LIN {X 0,Y 130.149,Z 483.599,A -85,B 0,C 180,E1 -28284.751,E2 -28284.751} C_VEL
LIN {X 0,Y 128.959,Z 485.397,A -85,B 0,C 180,E1 -28285.729,E2 -28285.729} C_VEL
LIN {X 0,Y 120.311,Z 494.144,A -85,B 0,C 180,E1 -28288.807,E2 -28288.807} C_VEL
LIN {X 0,Y 110.679,Z 502.592,A -85,B 0,C 180,E1 -28292.714,E2 -28292.714} C_VEL
LIN {X 0,Y 101.639,Z 509.611,A -85,B 0,C 180,E1 -28297.325,E2 -28297.325} C_VEL
LIN {X 0,Y 92.583,Z 515.883,A -85,B 0,C 180,E1 -28303.336,E2 -28303.336} C_VEL
LIN {X 0,Y 84.526,Z 520.929,A -85,B 0,C 180,E1 -28310.77,E2 -28310.77} C_VEL
LIN {X 0,Y 81.105,Z 522.68,A -85,B 0,C 180,E1 -28313.879,E2 -28313.879} C_VEL
LIN {X 0,Y 74.401,Z 525.173,A -85,B 0,C 180,E1 -28318.954,E2 -28318.954} C_VEL
LIN {X 0,Y 69.318,Z 526.805,A -85,B 0,C 180,E1 -28323.682,E2 -28323.682} C_VEL
LIN {X 0,Y 66.499,Z 527.76,A -85,B 0,C 180,E1 -28328.01,E2 -28328.01} C_VEL
LIN {X 0,Y 65.882,Z 527.988,A -85,B 0,C 180,E1 -28329.615,E2 -28329.615} C_VEL
LIN {X 0,Y 64.073,Z 528.951,A -85,B 0,C 180,E1 -28337.325,E2 -28337.325} C_VEL
LIN {X 0,Y 63.109,Z 529.528,A -85,B 0,C 180,E1 -28349.997,E2 -28349.997} C_VEL
LIN {X 0,Y 64.071,Z 528.979,A -85,B 0,C 180,E1 -28362.67,E2 -28362.67} C_VEL
LIN {X 0,Y 67.407,Z 527.331,A -85,B 0,C 180,E1 -28374.645,E2 -28374.645} C_VEL
LIN {X 0,Y 73.03,Z 524.535,A -85,B 0,C 180,E1 -28385.265,E2 -28385.265} C_VEL
LIN {X 0,Y 80.719,Z 520.508,A -85,B 0,C 180,E1 -28394.147,E2 -28394.147} C_VEL
LIN {X 0,Y 89.779,Z 515.164,A -85,B 0,C 180,E1 -28401.515,E2 -28401.515} C_VEL
LIN {X 0,Y 100.079,Z 508.331,A -85,B 0,C 180,E1 -28407.423,E2 -28407.423} C_VEL
LIN {X 0,Y 111.151,Z 499.793,A -85,B 0,C 180,E1 -28412.273,E2 -28412.273} C_VEL
LIN {X 0,Y 119.919,Z 492.105,A -85,B 0,C 180,E1 -28415.281,E2 -28415.281} C_VEL
LIN {X 0,Y 124.065,Z 488.02,A -85,B 0,C 180,E1 -28416.638,E2 -28416.638} C_VEL
LIN {X 0,Y 125.032,Z 486.59,A -85,B 0,C 180,E1 -28417.702,E2 -28417.702} C_VEL
LIN {X 0,Y 125.654,Z 484.374,A -85,B 0,C 180,E1 -28420.391,E2 -28420.391} C_VEL
LIN {X 0,Y 126.101,Z 482.181,A -85,B 0,C 180,E1 -28423.819,E2 -28423.819} C_VEL
LIN {X 0,Y 126.419,Z 480.387,A -85,B 0,C 180,E1 -28427.151,E2 -28427.151} C_VEL
LIN {X 0,Y 126.751,Z 478.972,A -85,B 0,C 180,E1 -28430.424,E2 -28430.424} C_VEL
LIN {X 0,Y 127.15,Z 477.836,A -85,B 0,C 180,E1 -28434.208,E2 -28434.208} C_VEL
LIN {X 0,Y 127.894,Z 476.973,A -85,B 0,C 180,E1 -28440,E2 -28440} C_VEL
LIN {X 0,Y 127.63,Z 477.823,A -85,B 0,C 180,E1 -28443.156,E2 -28443.156} C_VEL
LIN {X 0,Y 127.297,Z 479.151,A -85,B 0,C 180,E1 -28446.411,E2 -28446.411} C_VEL
LIN {X 0,Y 126.775,Z 480.998,A -85,B 0,C 180,E1 -28449.573,E2 -28449.573} C_VEL
LIN {X 0,Y 125.931,Z 483.628,A -85,B 0,C 180,E1 -28452.899,E2 -28452.899} C_VEL
LIN {X 0,Y 124.857,Z 486.8,A -85,B 0,C 180,E1 -28456.346,E2 -28456.346} C_VEL
LIN {X 0,Y 123.396,Z 490.697,A -85,B 0,C 180,E1 -28459.982,E2 -28459.982} C_VEL
LIN {X 0,Y 121.154,Z 493.836,A -85,B 0,C 180,E1 -28461.858,E2 -28461.858} C_VEL
LIN {X 0,Y 112.191,Z 502.139,A -85,B 0,C 180,E1 -28464.729,E2 -28464.729} C_VEL
LIN {X 0,Y 103.535,Z 509.243,A -85,B 0,C 180,E1 -28468.065,E2 -28468.065} C_VEL
LIN {X 0,Y 92.735,Z 517.125,A -85,B 0,C 180,E1 -28473.528,E2 -28473.528} C_VEL
LIN {X 0,Y 82.856,Z 523.405,A -85,B 0,C 180,E1 -28480.239,E2 -28480.239} C_VEL
LIN {X 0,Y 73.58,Z 528.827,A -85,B 0,C 180,E1 -28489.828,E2 -28489.828} C_VEL
LIN {X 0,Y 68.028,Z 531.891,A -85,B 0,C 180,E1 -28498.902,E2 -28498.902} C_VEL
LIN {X 0,Y 63.951,Z 534.284,A -85,B 0,C 180,E1 -28510.753,E2 -28510.753} C_VEL
LIN {X 0,Y 62.616,Z 535.521,A -85,B 0,C 180,E1 -28523.558,E2 -28523.558} C_VEL
LIN {X 0,Y 62.844,Z 535.701,A -85,B 0,C 180,E1 -28530.003,E2 -28530.003} C_VEL
LIN {X 0,Y 62.959,Z 535.026,A -85,B 0,C 180,E1 -28542.903,E2 -28542.903} C_VEL
LIN {X 0,Y 65.625,Z 533.183,A -85,B 0,C 180,E1 -28555.367,E2 -28555.367} C_VEL
LIN {X 0,Y 70.963,Z 530.169,A -85,B 0,C 180,E1 -28566.46,E2 -28566.46} C_VEL
LIN {X 0,Y 78.454,Z 525.917,A -85,B 0,C 180,E1 -28575.782,E2 -28575.782} C_VEL
LIN {X 0,Y 87.629,Z 520.319,A -85,B 0,C 180,E1 -28583.327,E2 -28583.327} C_VEL
LIN {X 0,Y 98.045,Z 513.228,A -85,B 0,C 180,E1 -28589.34,E2 -28589.34} C_VEL
LIN {X 0,Y 107.812,Z 505.657,A -85,B 0,C 180,E1 -28593.683,E2 -28593.683} C_VEL
LIN {X 0,Y 118.2,Z 496.56,A -85,B 0,C 180,E1 -28597.166,E2 -28597.166} C_VEL
LIN {X 0,Y 121.117,Z 493.584,A -85,B 0,C 180,E1 -28598.194,E2 -28598.194} C_VEL
LIN {X 0,Y 123.249,Z 490.578,A -85,B 0,C 180,E1 -28599.993,E2 -28599.993} C_VEL
LIN {X 0,Y 124.755,Z 486.626,A -85,B 0,C 180,E1 -28603.64,E2 -28603.64} C_VEL
LIN {X 0,Y 125.861,Z 483.397,A -85,B 0,C 180,E1 -28607.094,E2 -28607.094} C_VEL
LIN {X 0,Y 126.654,Z 480.815,A -85,B 0,C 180,E1 -28610.418,E2 -28610.418} C_VEL
LIN {X 0,Y 127.219,Z 478.794,A -85,B 0,C 180,E1 -28613.934,E2 -28613.934} C_VEL
LIN {X 0,Y 127.498,Z 477.621,A -85,B 0,C 180,E1 -28616.84,E2 -28616.84} C_VEL
LIN {X 0,Y 127.829,Z 476.691,A -85,B 0,C 180,E1 -28620,E2 -28620} C_VEL
LIN {X 0,Y 126.994,Z 477.733,A -85,B 0,C 180,E1 -28626.355,E2 -28626.355} C_VEL
LIN {X 0,Y 126.654,Z 478.731,A -85,B 0,C 180,E1 -28629.583,E2 -28629.583} C_VEL
LIN {X 0,Y 125.995,Z 481.959,A -85,B 0,C 180,E1 -28636.195,E2 -28636.195} C_VEL
LIN {X 0,Y 125.509,Z 484.19,A -85,B 0,C 180,E1 -28639.632,E2 -28639.632} C_VEL
LIN {X 0,Y 125.036,Z 486.267,A -85,B 0,C 180,E1 -28642.297,E2 -28642.297} C_VEL
LIN {X 0,Y 124.193,Z 487.599,A -85,B 0,C 180,E1 -28643.337,E2 -28643.337} C_VEL
LIN {X 0,Y 115.581,Z 495.835,A -85,B 0,C 180,E1 -28646.245,E2 -28646.245} C_VEL
LIN {X 0,Y 105.604,Z 504.046,A -85,B 0,C 180,E1 -28650.097,E2 -28650.097} C_VEL
LIN {X 0,Y 94.874,Z 511.747,A -85,B 0,C 180,E1 -28655.425,E2 -28655.425} C_VEL
LIN {X 0,Y 85.125,Z 517.861,A -85,B 0,C 180,E1 -28662.005,E2 -28662.005} C_VEL
LIN {X 0,Y 76.699,Z 522.566,A -85,B 0,C 180,E1 -28670.1,E2 -28670.1} C_VEL
LIN {X 0,Y 70.043,Z 525.994,A -85,B 0,C 180,E1 -28679.885,E2 -28679.885} C_VEL
LIN {X 0,Y 65.882,Z 527.988,A -85,B 0,C 180,E1 -28689.615,E2 -28689.615} C_VEL
LIN {X 0,Y 63.915,Z 528.739,A -85,B 0,C 180,E1 -28694.49,E2 -28694.49} C_VEL
LIN {X 0,Y 59.807,Z 529.608,A -85,B 0,C 180,E1 -28702.819,E2 -28702.819} C_VEL
LIN {X 0,Y 57.098,Z 529.875,A -85,B 0,C 180,E1 -28710.22,E2 -28710.22} C_VEL
LIN {X 0,Y 56.279,Z 529.774,A -85,B 0,C 180,E1 -28716.214,E2 -28716.214} C_VEL
LIN {X 0,Y 56.351,Z 529.675,A -85,B 0,C 180,E1 -28718.24,E2 -28718.24} C_VEL
LIN {X 0,Y 58.728,Z 528.644,A -85,B 0,C 180,E1 -28731.036,E2 -28731.036} C_VEL
LIN {X 0,Y 63.898,Z 526.429,A -85,B 0,C 180,E1 -28743.359,E2 -28743.359} C_VEL
LIN {X 0,Y 71.356,Z 523.027,A -85,B 0,C 180,E1 -28753.583,E2 -28753.583} C_VEL
LIN {X 0,Y 80.461,Z 518.361,A -85,B 0,C 180,E1 -28761.821,E2 -28761.821} C_VEL
LIN {X 0,Y 90.886,Z 512.291,A -85,B 0,C 180,E1 -28768.273,E2 -28768.273} C_VEL
LIN {X 0,Y 102.168,Z 504.637,A -85,B 0,C 180,E1 -28773.408,E2 -28773.408} C_VEL
LIN {X 0,Y 112.584,Z 496.465,A -85,B 0,C 180,E1 -28777.034,E2 -28777.034} C_VEL
LIN {X 0,Y 118.177,Z 491.487,A -85,B 0,C 180,E1 -28778.776,E2 -28778.776} C_VEL
LIN {X 0,Y 119.678,Z 489.96,A -85,B 0,C 180,E1 -28779.369,E2 -28779.369} C_VEL
LIN {X 0,Y 120.549,Z 487.505,A -85,B 0,C 180,E1 -28783.052,E2 -28783.052} C_VEL
LIN {X 0,Y 121.038,Z 485.65,A -85,B 0,C 180,E1 -28786.57,E2 -28786.57} C_VEL
LIN {X 0,Y 121.526,Z 484.182,A -85,B 0,C 180,E1 -28790.009,E2 -28790.009} C_VEL
LIN {X 0,Y 121.964,Z 483.164,A -85,B 0,C 180,E1 -28793.382,E2 -28793.382} C_VEL
LIN {X 0,Y 122.39,Z 482.492,A -85,B 0,C 180,E1 -28796.708,E2 -28796.708} C_VEL
LIN {X 0,Y 122.918,Z 482.094,A -85,B 0,C 180,E1 -28800,E2 -28800} C_VEL
LIN {X 0,Y 122.548,Z 483.015,A -85,B 0,C 180,E1 -28803.287,E2 -28803.287} C_VEL
LIN {X 0,Y 122.073,Z 484.429,A -85,B 0,C 180,E1 -28806.612,E2 -28806.612} C_VEL
LIN {X 0,Y 121.333,Z 486.432,A -85,B 0,C 180,E1 -28810.045,E2 -28810.045} C_VEL
LIN {X 0,Y 120.171,Z 489.211,A -85,B 0,C 180,E1 -28813.528,E2 -28813.528} C_VEL
LIN {X 0,Y 118.205,Z 493.414,A -85,B 0,C 180,E1 -28817.96,E2 -28817.96} C_VEL
LIN {X 0,Y 117.085,Z 494.983,A -85,B 0,C 180,E1 -28819.027,E2 -28819.027} C_VEL
LIN {X 0,Y 109.385,Z 501.789,A -85,B 0,C 180,E1 -28821.315,E2 -28821.315} C_VEL
LIN {X 0,Y 98.24,Z 510.432,A -85,B 0,C 180,E1 -28825.29,E2 -28825.29} C_VEL
LIN {X 0,Y 88.956,Z 516.773,A -85,B 0,C 180,E1 -28829.654,E2 -28829.654} C_VEL
LIN {X 0,Y 78.413,Z 523.055,A -85,B 0,C 180,E1 -28836.234,E2 -28836.234} C_VEL
LIN {X 0,Y 69.246,Z 527.938,A -85,B 0,C 180,E1 -28844.732,E2 -28844.732} C_VEL
LIN {X 0,Y 61.981,Z 531.539,A -85,B 0,C 180,E1 -28855.466,E2 -28855.466} C_VEL
LIN {X 0,Y 57.232,Z 533.933,A -85,B 0,C 180,E1 -28868.387,E2 -28868.387} C_VEL
LIN {X 0,Y 55.537,Z 535.172,A -85,B 0,C 180,E1 -28882.733,E2 -28882.733} C_VEL
LIN {X 0,Y 55.744,Z 535.353,A -85,B 0,C 180,E1 -28890.003,E2 -28890.003} C_VEL
LIN {X 0,Y 56.011,Z 534.675,A -85,B 0,C 180,E1 -28904.537,E2 -28904.537} C_VEL
LIN {X 0,Y 59.231,Z 532.831,A -85,B 0,C 180,E1 -28918.337,E2 -28918.337} C_VEL
LIN {X 0,Y 65.32,Z 529.816,A -85,B 0,C 180,E1 -28930.211,E2 -28930.211} C_VEL
LIN {X 0,Y 73.619,Z 525.563,A -85,B 0,C 180,E1 -28939.796,E2 -28939.796} C_VEL
LIN {X 0,Y 83.546,Z 519.966,A -85,B 0,C 180,E1 -28947.273,E2 -28947.273} C_VEL
LIN {X 0,Y 94.571,Z 512.873,A -85,B 0,C 180,E1 -28953.101,E2 -28953.101} C_VEL
LIN {X 0,Y 104.828,Z 505.304,A -85,B 0,C 180,E1 -28957.201,E2 -28957.201} C_VEL
LIN {X 0,Y 115.601,Z 496.205,A -85,B 0,C 180,E1 -28960.45,E2 -28960.45} C_VEL
LIN {X 0,Y 116.697,Z 495.146,A -85,B 0,C 180,E1 -28960.814,E2 -28960.814} C_VEL
LIN {X 0,Y 118.145,Z 493.152,A -85,B 0,C 180,E1 -28962.139,E2 -28962.139} C_VEL
LIN {X 0,Y 120.059,Z 489.041,A -85,B 0,C 180,E1 -28966.459,E2 -28966.459} C_VEL
LIN {X 0,Y 121.263,Z 486.123,A -85,B 0,C 180,E1 -28970.158,E2 -28970.158} C_VEL
LIN {X 0,Y 121.941,Z 484.262,A -85,B 0,C 180,E1 -28973.381,E2 -28973.381} C_VEL
LIN {X 0,Y 122.44,Z 482.805,A -85,B 0,C 180,E1 -28976.71,E2 -28976.71} C_VEL
LIN {X 0,Y 122.85,Z 481.837,A -85,B 0,C 180,E1 -28980,E2 -28980} C_VEL
LIN {X 0,Y 121.917,Z 482.897,A -85,B 0,C 180,E1 -28986.621,E2 -28986.621} C_VEL
LIN {X 0,Y 121.387,Z 484.041,A -85,B 0,C 180,E1 -28990.173,E2 -28990.173} C_VEL
LIN {X 0,Y 120.918,Z 485.447,A -85,B 0,C 180,E1 -28993.444,E2 -28993.444} C_VEL
LIN {X 0,Y 120.448,Z 487.299,A -85,B 0,C 180,E1 -28996.963,E2 -28996.963} C_VEL
LIN {X 0,Y 119.642,Z 489.695,A -85,B 0,C 180,E1 -29000.638,E2 -29000.638} C_VEL
LIN {X 0,Y 117.119,Z 492.213,A -85,B 0,C 180,E1 -29001.618,E2 -29001.618} C_VEL
LIN {X 0,Y 106.619,Z 501.083,A -85,B 0,C 180,E1 -29004.989,E2 -29004.989} C_VEL
LIN {X 0,Y 96.488,Z 508.459,A -85,B 0,C 180,E1 -29009.063,E2 -29009.063} C_VEL
LIN {X 0,Y 85.611,Z 515.339,A -85,B 0,C 180,E1 -29014.819,E2 -29014.819} C_VEL
LIN {X 0,Y 75.836,Z 520.726,A -85,B 0,C 180,E1 -29022.147,E2 -29022.147} C_VEL
LIN {X 0,Y 67.397,Z 524.784,A -85,B 0,C 180,E1 -29031.266,E2 -29031.266} C_VEL
LIN {X 0,Y 61.043,Z 527.614,A -85,B 0,C 180,E1 -29042.576,E2 -29042.576} C_VEL
LIN {X 0,Y 57.181,Z 529.298,A -85,B 0,C 180,E1 -29055.767,E2 -29055.767} C_VEL
LIN {X 0,Y 56.028,Z 529.875,A -85,B 0,C 180,E1 -29069.997,E2 -29069.997} C_VEL
LIN {X 0,Y 56.351,Z 529.675,A -85,B 0,C 180,E1 -29078.24,E2 -29078.24} C_VEL
LIN {X 0,Y 56.46,Z 529.382,A -85,B 0,C 180,E1 -29084.229,E2 -29084.229} C_VEL
LIN {X 0,Y 56.059,Z 528.599,A -85,B 0,C 180,E1 -29094.306,E2 -29094.306} C_VEL
LIN {X 0,Y 56.713,Z 527.628,A -85,B 0,C 180,E1 -29102.34,E2 -29102.34} C_VEL
LIN {X 0,Y 58.558,Z 526.611,A -85,B 0,C 180,E1 -29107.867,E2 -29107.867} C_VEL
LIN {X 0,Y 59.507,Z 526.179,A -85,B 0,C 180,E1 -29109.509,E2 -29109.509} C_VEL
LIN {X 0,Y 68.747,Z 522.331,A -85,B 0,C 180,E1 -29120.056,E2 -29120.056} C_VEL
LIN {X 0,Y 78.615,Z 517.476,A -85,B 0,C 180,E1 -29127.561,E2 -29127.561} C_VEL
LIN {X 0,Y 90.254,Z 510.856,A -85,B 0,C 180,E1 -29133.568,E2 -29133.568} C_VEL
LIN {X 0,Y 100.712,Z 503.88,A -85,B 0,C 180,E1 -29137.607,E2 -29137.607} C_VEL
LIN {X 0,Y 110.009,Z 496.811,A -85,B 0,C 180,E1 -29140.438,E2 -29140.438} C_VEL
LIN {X 0,Y 113.254,Z 494.029,A -85,B 0,C 180,E1 -29141.363,E2 -29141.363} C_VEL
LIN {X 0,Y 114.627,Z 492.7,A -85,B 0,C 180,E1 -29142.148,E2 -29142.148} C_VEL
LIN {X 0,Y 115.551,Z 490.344,A -85,B 0,C 180,E1 -29146.685,E2 -29146.685} C_VEL
LIN {X 0,Y 116.039,Z 489.208,A -85,B 0,C 180,E1 -29149.531,E2 -29149.531} C_VEL
LIN {X 0,Y 116.646,Z 488.115,A -85,B 0,C 180,E1 -29153.079,E2 -29153.079} C_VEL
LIN {X 0,Y 117.14,Z 487.416,A -85,B 0,C 180,E1 -29156.56,E2 -29156.56} C_VEL
LIN {X 0,Y 117.71,Z 487.034,A -85,B 0,C 180,E1 -29160,E2 -29160} C_VEL
LIN {X 0,Y 117.222,Z 488.024,A -85,B 0,C 180,E1 -29163.437,E2 -29163.437} C_VEL
LIN {X 0,Y 116.549,Z 489.569,A -85,B 0,C 180,E1 -29166.926,E2 -29166.926} C_VEL
LIN {X 0,Y 115.876,Z 490.999,A -85,B 0,C 180,E1 -29169.46,E2 -29169.46} C_VEL
LIN {X 0,Y 114.413,Z 493.75,A -85,B 0,C 180,E1 -29173.088,E2 -29173.088} C_VEL
LIN {X 0,Y 112.922,Z 496.405,A -85,B 0,C 180,E1 -29176.088,E2 -29176.088} C_VEL
LIN {X 0,Y 110.192,Z 498.818,A -85,B 0,C 180,E1 -29176.929,E2 -29176.929} C_VEL
LIN {X 0,Y 99.142,Z 507.411,A -85,B 0,C 180,E1 -29180.076,E2 -29180.076} C_VEL
LIN {X 0,Y 88.566,Z 514.585,A -85,B 0,C 180,E1 -29184.143,E2 -29184.143} C_VEL
LIN {X 0,Y 77.098,Z 521.252,A -85,B 0,C 180,E1 -29190.009,E2 -29190.009} C_VEL
LIN {X 0,Y 66.741,Z 526.491,A -85,B 0,C 180,E1 -29197.84,E2 -29197.84} C_VEL
LIN {X 0,Y 60.028,Z 529.541,A -85,B 0,C 180,E1 -29205.378,E2 -29205.378} C_VEL
LIN {X 0,Y 53.032,Z 532.531,A -85,B 0,C 180,E1 -29217.992,E2 -29217.992} C_VEL
LIN {X 0,Y 49.123,Z 534.346,A -85,B 0,C 180,E1 -29233.377,E2 -29233.377} C_VEL
LIN {X 0,Y 48.635,Z 535.005,A -85,B 0,C 180,E1 -29250.004,E2 -29250.004} C_VEL
LIN {X 0,Y 49.133,Z 534.325,A -85,B 0,C 180,E1 -29266.627,E2 -29266.627} C_VEL
LIN {X 0,Y 53.037,Z 532.48,A -85,B 0,C 180,E1 -29282.012,E2 -29282.012} C_VEL
LIN {X 0,Y 60.002,Z 529.463,A -85,B 0,C 180,E1 -29294.654,E2 -29294.654} C_VEL
LIN {X 0,Y 69.188,Z 525.209,A -85,B 0,C 180,E1 -29304.357,E2 -29304.357} C_VEL
LIN {X 0,Y 79.898,Z 519.613,A -85,B 0,C 180,E1 -29311.601,E2 -29311.601} C_VEL
LIN {X 0,Y 91.537,Z 512.518,A -85,B 0,C 180,E1 -29317.127,E2 -29317.127} C_VEL
LIN {X 0,Y 102.264,Z 504.95,A -85,B 0,C 180,E1 -29320.905,E2 -29320.905} C_VEL
LIN {X 0,Y 111.581,Z 497.405,A -85,B 0,C 180,E1 -29323.418,E2 -29323.418} C_VEL
LIN {X 0,Y 112.858,Z 496.205,A -85,B 0,C 180,E1 -29323.947,E2 -29323.947} C_VEL
LIN {X 0,Y 114.878,Z 492.523,A -85,B 0,C 180,E1 -29328.202,E2 -29328.202} C_VEL
LIN {X 0,Y 115.837,Z 490.697,A -85,B 0,C 180,E1 -29330.743,E2 -29330.743} C_VEL
LIN {X 0,Y 116.432,Z 489.399,A -85,B 0,C 180,E1 -29333.067,E2 -29333.067} C_VEL
LIN {X 0,Y 117.127,Z 487.82,A -85,B 0,C 180,E1 -29336.56,E2 -29336.56} C_VEL
LIN {X 0,Y 117.647,Z 486.796,A -85,B 0,C 180,E1 -29340,E2 -29340} C_VEL
LIN {X 0,Y 117.101,Z 487.15,A -85,B 0,C 180,E1 -29343.441,E2 -29343.441} C_VEL
LIN {X 0,Y 116.533,Z 487.94,A -85,B 0,C 180,E1 -29347.127,E2 -29347.127} C_VEL
LIN {X 0,Y 115.942,Z 489.007,A -85,B 0,C 180,E1 -29350.478,E2 -29350.478} C_VEL
LIN {X 0,Y 115.285,Z 490.524,A -85,B 0,C 180,E1 -29354.114,E2 -29354.114} C_VEL
LIN {X 0,Y 114.57,Z 492.479,A -85,B 0,C 180,E1 -29357.862,E2 -29357.862} C_VEL
LIN {X 0,Y 113.209,Z 493.828,A -85,B 0,C 180,E1 -29358.721,E2 -29358.721} C_VEL
LIN {X 0,Y 102.284,Z 502.542,A -85,B 0,C 180,E1 -29361.933,E2 -29361.933} C_VEL
LIN {X 0,Y 93.241,Z 508.809,A -85,B 0,C 180,E1 -29365.241,E2 -29365.241} C_VEL
LIN {X 0,Y 81.752,Z 515.69,A -85,B 0,C 180,E1 -29370.717,E2 -29370.717} C_VEL
LIN {X 0,Y 71.256,Z 521.076,A -85,B 0,C 180,E1 -29377.9,E2 -29377.9} C_VEL
LIN {X 0,Y 61.998,Z 525.135,A -85,B 0,C 180,E1 -29387.141,E2 -29387.141} C_VEL
LIN {X 0,Y 54.835,Z 527.962,A -85,B 0,C 180,E1 -29399.155,E2 -29399.155} C_VEL
LIN {X 0,Y 50.326,Z 529.646,A -85,B 0,C 180,E1 -29413.778,E2 -29413.778} C_VEL
LIN {X 0,Y 48.948,Z 530.222,A -85,B 0,C 180,E1 -29429.997,E2 -29429.997} C_VEL
LIN {X 0,Y 50.323,Z 529.674,A -85,B 0,C 180,E1 -29446.216,E2 -29446.216} C_VEL
LIN {X 0,Y 54.804,Z 528.027,A -85,B 0,C 180,E1 -29460.857,E2 -29460.857} C_VEL
LIN {X 0,Y 59.507,Z 526.179,A -85,B 0,C 180,E1 -29469.509,E2 -29469.509} C_VEL
LIN {X 0,Y 62.237,Z 524.952,A -85,B 0,C 180,E1 -29474.31,E2 -29474.31} C_VEL
LIN {X 0,Y 66.129,Z 522.653,A -85,B 0,C 180,E1 -29482.231,E2 -29482.231} C_VEL
LIN {X 0,Y 69.864,Z 520.508,A -85,B 0,C 180,E1 -29487.876,E2 -29487.876} C_VEL
LIN {X 0,Y 73.552,Z 518.573,A -85,B 0,C 180,E1 -29491.239,E2 -29491.239} C_VEL
LIN {X 0,Y 74.987,Z 517.842,A -85,B 0,C 180,E1 -29492.122,E2 -29492.122} C_VEL
LIN {X 0,Y 87.321,Z 511.203,A -85,B 0,C 180,E1 -29497.75,E2 -29497.75} C_VEL
LIN {X 0,Y 98.214,Z 504.229,A -85,B 0,C 180,E1 -29501.462,E2 -29501.462} C_VEL
LIN {X 0,Y 108.163,Z 496.888,A -85,B 0,C 180,E1 -29504.085,E2 -29504.085} C_VEL
LIN {X 0,Y 109.307,Z 495.847,A -85,B 0,C 180,E1 -29504.668,E2 -29504.668} C_VEL
LIN {X 0,Y 110.32,Z 494.018,A -85,B 0,C 180,E1 -29508.982,E2 -29508.982} C_VEL
LIN {X 0,Y 111.063,Z 492.878,A -85,B 0,C 180,E1 -29512.729,E2 -29512.729} C_VEL
LIN {X 0,Y 111.686,Z 492.126,A -85,B 0,C 180,E1 -29516.392,E2 -29516.392} C_VEL
LIN {X 0,Y 112.3,Z 491.762,A -85,B 0,C 180,E1 -29520,E2 -29520} C_VEL
LIN {X 0,Y 111.666,Z 492.827,A -85,B 0,C 180,E1 -29523.608,E2 -29523.608} C_VEL
LIN {X 0,Y 110.768,Z 494.493,A -85,B 0,C 180,E1 -29527.29,E2 -29527.29} C_VEL
LIN {X 0,Y 109.203,Z 496.948,A -85,B 0,C 180,E1 -29531.132,E2 -29531.132} C_VEL
LIN {X 0,Y 108.206,Z 498.444,A -85,B 0,C 180,E1 -29533.036,E2 -29533.036} C_VEL
LIN {X 0,Y 106.676,Z 499.832,A -85,B 0,C 180,E1 -29533.657,E2 -29533.657} C_VEL
LIN {X 0,Y 95.317,Z 508.193,A -85,B 0,C 180,E1 -29536.565,E2 -29536.565} C_VEL
LIN {X 0,Y 82.785,Z 516.07,A -85,B 0,C 180,E1 -29540.965,E2 -29540.965} C_VEL
LIN {X 0,Y 70.864,Z 522.352,A -85,B 0,C 180,E1 -29546.806,E2 -29546.806} C_VEL
LIN {X 0,Y 60.01,Z 527.235,A -85,B 0,C 180,E1 -29554.941,E2 -29554.941} C_VEL
LIN {X 0,Y 50.794,Z 530.835,A -85,B 0,C 180,E1 -29566.231,E2 -29566.231} C_VEL
LIN {X 0,Y 44.202,Z 533.23,A -85,B 0,C 180,E1 -29581.516,E2 -29581.516} C_VEL
LIN {X 0,Y 41.416,Z 534.472,A -85,B 0,C 180,E1 -29600.234,E2 -29600.234} C_VEL
LIN {X 0,Y 41.523,Z 534.656,A -85,B 0,C 180,E1 -29610.004,E2 -29610.004} C_VEL
LIN {X 0,Y 42.318,Z 533.974,A -85,B 0,C 180,E1 -29629.404,E2 -29629.404} C_VEL
LIN {X 0,Y 47.12,Z 532.128,A -85,B 0,C 180,E1 -29646.632,E2 -29646.632} C_VEL
LIN {X 0,Y 56.558,Z 528.547,A -85,B 0,C 180,E1 -29661.589,E2 -29661.589} C_VEL
LIN {X 0,Y 68.04,Z 523.587,A -85,B 0,C 180,E1 -29671.404,E2 -29671.404} C_VEL
LIN {X 0,Y 79.751,Z 517.618,A -85,B 0,C 180,E1 -29677.719,E2 -29677.719} C_VEL
LIN {X 0,Y 92.159,Z 510.1,A -85,B 0,C 180,E1 -29682.48,E2 -29682.48} C_VEL
LIN {X 0,Y 103.404,Z 502.119,A -85,B 0,C 180,E1 -29685.593,E2 -29685.593} C_VEL
LIN {X 0,Y 106.685,Z 499.599,A -85,B 0,C 180,E1 -29686.337,E2 -29686.337} C_VEL
LIN {X 0,Y 108.173,Z 498.198,A -85,B 0,C 180,E1 -29687.053,E2 -29687.053} C_VEL
LIN {X 0,Y 110.022,Z 495.416,A -85,B 0,C 180,E1 -29690.811,E2 -29690.811} C_VEL
LIN {X 0,Y 110.681,Z 494.311,A -85,B 0,C 180,E1 -29692.704,E2 -29692.704} C_VEL
LIN {X 0,Y 111.551,Z 492.659,A -85,B 0,C 180,E1 -29696.388,E2 -29696.388} C_VEL
LIN {X 0,Y 112.241,Z 491.542,A -85,B 0,C 180,E1 -29700,E2 -29700} C_VEL
LIN {X 0,Y 111.657,Z 491.876,A -85,B 0,C 180,E1 -29703.609,E2 -29703.609} C_VEL
LIN {X 0,Y 110.999,Z 492.653,A -85,B 0,C 180,E1 -29707.275,E2 -29707.275} C_VEL
LIN {X 0,Y 110.252,Z 493.812,A -85,B 0,C 180,E1 -29711.025,E2 -29711.025} C_VEL
LIN {X 0,Y 109.256,Z 495.589,A -85,B 0,C 180,E1 -29715.221,E2 -29715.221} C_VEL
LIN {X 0,Y 108.121,Z 496.679,A -85,B 0,C 180,E1 -29715.993,E2 -29715.993} C_VEL
LIN {X 0,Y 96.691,Z 505.096,A -85,B 0,C 180,E1 -29719.103,E2 -29719.103} C_VEL
LIN {X 0,Y 84.313,Z 512.798,A -85,B 0,C 180,E1 -29723.517,E2 -29723.517} C_VEL
LIN {X 0,Y 72.59,Z 518.911,A -85,B 0,C 180,E1 -29729.378,E2 -29729.378} C_VEL
LIN {X 0,Y 61.887,Z 523.613,A -85,B 0,C 180,E1 -29737.347,E2 -29737.347} C_VEL
LIN {X 0,Y 52.65,Z 527.044,A -85,B 0,C 180,E1 -29748.127,E2 -29748.127} C_VEL
LIN {X 0,Y 45.768,Z 529.294,A -85,B 0,C 180,E1 -29762.565,E2 -29762.565} C_VEL
LIN {X 0,Y 42.243,Z 530.422,A -85,B 0,C 180,E1 -29780.419,E2 -29780.419} C_VEL
LIN {X 0,Y 41.857,Z 530.569,A -85,B 0,C 180,E1 -29789.996,E2 -29789.996} C_VEL
LIN {X 0,Y 43.564,Z 530.021,A -85,B 0,C 180,E1 -29808.819,E2 -29808.819} C_VEL
LIN {X 0,Y 48.832,Z 528.375,A -85,B 0,C 180,E1 -29825.143,E2 -29825.143} C_VEL
LIN {X 0,Y 56.931,Z 525.58,A -85,B 0,C 180,E1 -29837.786,E2 -29837.786} C_VEL
LIN {X 0,Y 67.051,Z 521.553,A -85,B 0,C 180,E1 -29846.98,E2 -29846.98} C_VEL
LIN {X 0,Y 74.987,Z 517.842,A -85,B 0,C 180,E1 -29852.122,E2 -29852.122} C_VEL
LIN {X 0,Y 79.114,Z 515.657,A -85,B 0,C 180,E1 -29854.805,E2 -29854.805} C_VEL
LIN {X 0,Y 85.182,Z 511.902,A -85,B 0,C 180,E1 -29859.624,E2 -29859.624} C_VEL
LIN {X 0,Y 91.527,Z 507.713,A -85,B 0,C 180,E1 -29863.758,E2 -29863.758} C_VEL
LIN {X 0,Y 95.89,Z 504.777,A -85,B 0,C 180,E1 -29865.408,E2 -29865.408} C_VEL
LIN {X 0,Y 103.099,Z 499.717,A -85,B 0,C 180,E1 -29867.088,E2 -29867.088} C_VEL
LIN {X 0,Y 104.277,Z 498.669,A -85,B 0,C 180,E1 -29868.334,E2 -29868.334} C_VEL
LIN {X 0,Y 105.255,Z 497.421,A -85,B 0,C 180,E1 -29872.325,E2 -29872.325} C_VEL
LIN {X 0,Y 106.029,Z 496.62,A -85,B 0,C 180,E1 -29876.199,E2 -29876.199} C_VEL
LIN {X 0,Y 106.676,Z 496.285,A -85,B 0,C 180,E1 -29880,E2 -29880} C_VEL
LIN {X 0,Y 105.706,Z 497.635,A -85,B 0,C 180,E1 -29884.237,E2 -29884.237} C_VEL
LIN {X 0,Y 104.625,Z 499.277,A -85,B 0,C 180,E1 -29887.72,E2 -29887.72} C_VEL
LIN {X 0,Y 103.478,Z 500.728,A -85,B 0,C 180,E1 -29890.008,E2 -29890.008} C_VEL
LIN {X 0,Y 100.172,Z 503.23,A -85,B 0,C 180,E1 -29890.826,E2 -29890.826} C_VEL
LIN {X 0,Y 87.429,Z 511.693,A -85,B 0,C 180,E1 -29893.954,E2 -29893.954} C_VEL
LIN {X 0,Y 74.146,Z 519.047,A -85,B 0,C 180,E1 -29898.591,E2 -29898.591} C_VEL
LIN {X 0,Y 61.929,Z 524.608,A -85,B 0,C 180,E1 -29904.793,E2 -29904.793} C_VEL
LIN {X 0,Y 50.808,Z 528.838,A -85,B 0,C 180,E1 -29913.913,E2 -29913.913} C_VEL
LIN {X 0,Y 41.573,Z 531.829,A -85,B 0,C 180,E1 -29927.458,E2 -29927.458} C_VEL
LIN {X 0,Y 35.642,Z 533.645,A -85,B 0,C 180,E1 -29946.779,E2 -29946.779} C_VEL
LIN {X 0,Y 34.405,Z 534.307,A -85,B 0,C 180,E1 -29970.005,E2 -29970.005} C_VEL
LIN {X 0,Y 35.65,Z 533.623,A -85,B 0,C 180,E1 -29993.226,E2 -29993.226} C_VEL
LIN {X 0,Y 41.574,Z 531.776,A -85,B 0,C 180,E1 -30012.552,E2 -30012.552} C_VEL
LIN {X 0,Y 51.639,Z 528.456,A -85,B 0,C 180,E1 -30027.018,E2 -30027.018} C_VEL
LIN {X 0,Y 61.925,Z 524.503,A -85,B 0,C 180,E1 -30035.228,E2 -30035.228} C_VEL
LIN {X 0,Y 74.151,Z 518.907,A -85,B 0,C 180,E1 -30041.411,E2 -30041.411} C_VEL
LIN {X 0,Y 87.434,Z 511.509,A -85,B 0,C 180,E1 -30046.047,E2 -30046.047} C_VEL
LIN {X 0,Y 100.181,Z 503.01,A -85,B 0,C 180,E1 -30049.164,E2 -30049.164} C_VEL
LIN {X 0,Y 101.861,Z 501.767,A -85,B 0,C 180,E1 -30049.489,E2 -30049.489} C_VEL
LIN {X 0,Y 103.451,Z 500.498,A -85,B 0,C 180,E1 -30050.095,E2 -30050.095} C_VEL
LIN {X 0,Y 104.574,Z 499.081,A -85,B 0,C 180,E1 -30052.276,E2 -30052.276} C_VEL
LIN {X 0,Y 105.731,Z 497.293,A -85,B 0,C 180,E1 -30056.189,E2 -30056.189} C_VEL
LIN {X 0,Y 106.621,Z 496.081,A -85,B 0,C 180,E1 -30060,E2 -30060} C_VEL
LIN {X 0,Y 105.787,Z 496.571,A -85,B 0,C 180,E1 -30064.756,E2 -30064.756} C_VEL
LIN {X 0,Y 105.197,Z 497.21,A -85,B 0,C 180,E1 -30067.679,E2 -30067.679} C_VEL
LIN {X 0,Y 104.236,Z 498.462,A -85,B 0,C 180,E1 -30071.67,E2 -30071.67} C_VEL
LIN {X 0,Y 103.067,Z 499.517,A -85,B 0,C 180,E1 -30072.998,E2 -30072.998} C_VEL
LIN {X 0,Y 91.348,Z 507.519,A -85,B 0,C 180,E1 -30075.901,E2 -30075.901} C_VEL
LIN {X 0,Y 78.593,Z 514.801,A -85,B 0,C 180,E1 -30080.121,E2 -30080.121} C_VEL
LIN {X 0,Y 66.395,Z 520.563,A -85,B 0,C 180,E1 -30085.87,E2 -30085.87} C_VEL
LIN {X 0,Y 57.854,Z 523.962,A -85,B 0,C 180,E1 -30091.746,E2 -30091.746} C_VEL
LIN {X 0,Y 47.591,Z 527.393,A -85,B 0,C 180,E1 -30102.401,E2 -30102.401} C_VEL
LIN {X 0,Y 39.604,Z 529.642,A -85,B 0,C 180,E1 -30117.829,E2 -30117.829} C_VEL
LIN {X 0,Y 35.276,Z 530.769,A -85,B 0,C 180,E1 -30138.503,E2 -30138.503} C_VEL
LIN {X 0,Y 34.775,Z 530.916,A -85,B 0,C 180,E1 -30149.995,E2 -30149.995} C_VEL
LIN {X 0,Y 36.901,Z 530.369,A -85,B 0,C 180,E1 -30172.385,E2 -30172.385} C_VEL
LIN {X 0,Y 43.203,Z 528.724,A -85,B 0,C 180,E1 -30190.589,E2 -30190.589} C_VEL
LIN {X 0,Y 52.412,Z 525.929,A -85,B 0,C 180,E1 -30203.561,E2 -30203.561} C_VEL
LIN {X 0,Y 63.445,Z 521.902,A -85,B 0,C 180,E1 -30212.392,E2 -30212.392} C_VEL
LIN {X 0,Y 75.43,Z 516.554,A -85,B 0,C 180,E1 -30218.698,E2 -30218.698} C_VEL
LIN {X 0,Y 88.079,Z 509.72,A -85,B 0,C 180,E1 -30223.23,E2 -30223.23} C_VEL
LIN {X 0,Y 95.89,Z 504.777,A -85,B 0,C 180,E1 -30225.408,E2 -30225.408} C_VEL
LIN {X 0,Y 97.555,Z 503.585,A -85,B 0,C 180,E1 -30226.243,E2 -30226.243} C_VEL
LIN {X 0,Y 98.909,Z 502.471,A -85,B 0,C 180,E1 -30227.805,E2 -30227.805} C_VEL
LIN {X 0,Y 99.807,Z 501.496,A -85,B 0,C 180,E1 -30230.39,E2 -30230.39} C_VEL
LIN {X 0,Y 100.074,Z 501.024,A -85,B 0,C 180,E1 -30233.87,E2 -30233.87} C_VEL
LIN {X 0,Y 100.34,Z 500.796,A -85,B 0,C 180,E1 -30237.361,E2 -30237.361} C_VEL
LIN {X 0,Y 100.831,Z 500.602,A -85,B 0,C 180,E1 -30240,E2 -30240} C_VEL
LIN {X 0,Y 99.744,Z 501.88,A -85,B 0,C 180,E1 -30244.04,E2 -30244.04} C_VEL
LIN {X 0,Y 98.985,Z 502.842,A -85,B 0,C 180,E1 -30246.293,E2 -30246.293} C_VEL
LIN {X 0,Y 97.367,Z 504.101,A -85,B 0,C 180,E1 -30247.047,E2 -30247.047} C_VEL
LIN {X 0,Y 85.1,Z 511.876,A -85,B 0,C 180,E1 -30249.507,E2 -30249.507} C_VEL
LIN {X 0,Y 72.178,Z 518.696,A -85,B 0,C 180,E1 -30253.179,E2 -30253.179} C_VEL
LIN {X 0,Y 59.277,Z 524.257,A -85,B 0,C 180,E1 -30258.479,E2 -30258.479} C_VEL
LIN {X 0,Y 47.182,Z 528.487,A -85,B 0,C 180,E1 -30266.662,E2 -30266.662} C_VEL
LIN {X 0,Y 36.609,Z 531.478,A -85,B 0,C 180,E1 -30279.843,E2 -30279.843} C_VEL
LIN {X 0,Y 29.183,Z 533.294,A -85,B 0,C 180,E1 -30301.213,E2 -30301.213} C_VEL
LIN {X 0,Y 27.279,Z 533.958,A -85,B 0,C 180,E1 -30330.006,E2 -30330.006} C_VEL
LIN {X 0,Y 29.191,Z 533.271,A -85,B 0,C 180,E1 -30358.791,E2 -30358.791} C_VEL
LIN {X 0,Y 36.609,Z 531.423,A -85,B 0,C 180,E1 -30380.172,E2 -30380.172} C_VEL
LIN {X 0,Y 47.306,Z 528.357,A -85,B 0,C 180,E1 -30393.533,E2 -30393.533} C_VEL
LIN {X 0,Y 59.278,Z 524.15,A -85,B 0,C 180,E1 -30401.537,E2 -30401.537} C_VEL
LIN {X 0,Y 72.183,Z 518.554,A -85,B 0,C 180,E1 -30406.823,E2 -30406.823} C_VEL
LIN {X 0,Y 85.492,Z 511.456,A -85,B 0,C 180,E1 -30410.578,E2 -30410.578} C_VEL
LIN {X 0,Y 97.375,Z 503.891,A -85,B 0,C 180,E1 -30412.945,E2 -30412.945} C_VEL
LIN {X 0,Y 98.977,Z 502.61,A -85,B 0,C 180,E1 -30413.781,E2 -30413.781} C_VEL
LIN {X 0,Y 99.652,Z 501.722,A -85,B 0,C 180,E1 -30415.956,E2 -30415.956} C_VEL
LIN {X 0,Y 100.768,Z 500.42,A -85,B 0,C 180,E1 -30420,E2 -30420} C_VEL
LIN {X 0,Y 100.144,Z 500.683,A -85,B 0,C 180,E1 -30424.025,E2 -30424.025} C_VEL
LIN {X 0,Y 99.12,Z 501.582,A -85,B 0,C 180,E1 -30428.153,E2 -30428.153} C_VEL
LIN {X 0,Y 98.001,Z 502.519,A -85,B 0,C 180,E1 -30429.747,E2 -30429.747} C_VEL
LIN {X 0,Y 86.325,Z 509.86,A -85,B 0,C 180,E1 -30432.315,E2 -30432.315} C_VEL
LIN {X 0,Y 73.181,Z 516.741,A -85,B 0,C 180,E1 -30436.179,E2 -30436.179} C_VEL
LIN {X 0,Y 60.517,Z 522.128,A -85,B 0,C 180,E1 -30441.705,E2 -30441.705} C_VEL
LIN {X 0,Y 48.561,Z 526.184,A -85,B 0,C 180,E1 -30449.726,E2 -30449.726} C_VEL
LIN {X 0,Y 38.118,Z 529.009,A -85,B 0,C 180,E1 -30462.475,E2 -30462.475} C_VEL
LIN {X 0,Y 30.453,Z 530.691,A -85,B 0,C 180,E1 -30482.505,E2 -30482.505} C_VEL
LIN {X 0,Y 27.696,Z 531.263,A -85,B 0,C 180,E1 -30509.994,E2 -30509.994} C_VEL
LIN {X 0,Y 30.448,Z 530.717,A -85,B 0,C 180,E1 -30537.487,E2 -30537.487} C_VEL
LIN {X 0,Y 38.084,Z 529.072,A -85,B 0,C 180,E1 -30557.567,E2 -30557.567} C_VEL
LIN {X 0,Y 48.521,Z 526.277,A -85,B 0,C 180,E1 -30570.343,E2 -30570.343} C_VEL
LIN {X 0,Y 60.464,Z 522.251,A -85,B 0,C 180,E1 -30578.407,E2 -30578.407} C_VEL
LIN {X 0,Y 73.144,Z 516.902,A -85,B 0,C 180,E1 -30583.905,E2 -30583.905} C_VEL
LIN {X 0,Y 86.297,Z 510.066,A -85,B 0,C 180,E1 -30587.751,E2 -30587.751} C_VEL
LIN {X 0,Y 98.03,Z 502.711,A -85,B 0,C 180,E1 -30590.34,E2 -30590.34} C_VEL
LIN {X 0,Y 99.291,Z 501.663,A -85,B 0,C 180,E1 -30592.272,E2 -30592.272} C_VEL
LIN {X 0,Y 100.169,Z 500.897,A -85,B 0,C 180,E1 -30595.976,E2 -30595.976} C_VEL
LIN {X 0,Y 100.34,Z 500.796,A -85,B 0,C 180,E1 -30597.361,E2 -30597.361} C_VEL
LIN {X 0,Y 99.88,Z 501.194,A -85,B 0,C 180,E1 -30598.938,E2 -30598.938} C_VEL
LIN {X 0,Y 98.118,Z 502.559,A -85,B 0,C 180,E1 -30600.587,E2 -30600.587} C_VEL
LIN {X 0,Y 95.394,Z 504.502,A -85,B 0,C 180,E1 -30601.977,E2 -30601.977} C_VEL
LIN {X 0,Y 90.603,Z 507.713,A -85,B 0,C 180,E1 -30603.445,E2 -30603.445} C_VEL
LIN {X 0,Y 85.466,Z 510.786,A -85,B 0,C 180,E1 -30604.487,E2 -30604.487} C_VEL
LIN {X 0,Y 74.298,Z 516.705,A -85,B 0,C 180,E1 -30606.696,E2 -30606.696} C_VEL
LIN {X 0,Y 60.741,Z 522.635,A -85,B 0,C 180,E1 -30610.441,E2 -30610.441} C_VEL
LIN {X 0,Y 50.828,Z 526.18,A -85,B 0,C 180,E1 -30614.572,E2 -30614.572} C_VEL
LIN {X 0,Y 38.264,Z 529.782,A -85,B 0,C 180,E1 -30623.324,E2 -30623.324} C_VEL
LIN {X 0,Y 27.289,Z 532.176,A -85,B 0,C 180,E1 -30639.42,E2 -30639.42} C_VEL
LIN {X 0,Y 20.628,Z 533.423,A -85,B 0,C 180,E1 -30670.089,E2 -30670.089} C_VEL
LIN {X 0,Y 20.173,Z 533.61,A -85,B 0,C 180,E1 -30690.008,E2 -30690.008} C_VEL
LIN {X 0,Y 23.163,Z 532.919,A -85,B 0,C 180,E1 -30727.37,E2 -30727.37} C_VEL
LIN {X 0,Y 32.486,Z 531.071,A -85,B 0,C 180,E1 -30749.932,E2 -30749.932} C_VEL
LIN {X 0,Y 44.408,Z 528.05,A -85,B 0,C 180,E1 -30761.735,E2 -30761.735} C_VEL
LIN {X 0,Y 57.409,Z 523.797,A -85,B 0,C 180,E1 -30768.353,E2 -30768.353} C_VEL
LIN {X 0,Y 70.892,Z 518.201,A -85,B 0,C 180,E1 -30772.481,E2 -30772.481} C_VEL
LIN {X 0,Y 84.615,Z 511.103,A -85,B 0,C 180,E1 -30775.371,E2 -30775.371} C_VEL
LIN {X 0,Y 91.54,Z 506.932,A -85,B 0,C 180,E1 -30776.476,E2 -30776.476} C_VEL
LIN {X 0,Y 93.954,Z 505.28,A -85,B 0,C 180,E1 -30777.425,E2 -30777.425} C_VEL
LIN {X 0,Y 94.703,Z 504.536,A -85,B 0,C 180,E1 -30780,E2 -30780} C_VEL
LIN {X 0,Y 93.773,Z 504.955,A -85,B 0,C 180,E1 -30785.305,E2 -30785.305} C_VEL
LIN {X 0,Y 91.947,Z 506.147,A -85,B 0,C 180,E1 -30786.439,E2 -30786.439} C_VEL
LIN {X 0,Y 78.282,Z 513.848,A -85,B 0,C 180,E1 -30789.036,E2 -30789.036} C_VEL
LIN {X 0,Y 64.837,Z 519.963,A -85,B 0,C 180,E1 -30792.682,E2 -30792.682} C_VEL
LIN {X 0,Y 51.793,Z 524.662,A -85,B 0,C 180,E1 -30798.212,E2 -30798.212} C_VEL
LIN {X 0,Y 39.421,Z 528.092,A -85,B 0,C 180,E1 -30806.939,E2 -30806.939} C_VEL
LIN {X 0,Y 28.588,Z 530.34,A -85,B 0,C 180,E1 -30822.471,E2 -30822.471} C_VEL
LIN {X 0,Y 21.55,Z 531.465,A -85,B 0,C 180,E1 -30850.958,E2 -30850.958} C_VEL
LIN {X 0,Y 20.616,Z 531.61,A -85,B 0,C 180,E1 -30869.992,E2 -30869.992} C_VEL
LIN {X 0,Y 24.375,Z 531.065,A -85,B 0,C 180,E1 -30905.207,E2 -30905.207} C_VEL
LIN {X 0,Y 33.701,Z 529.42,A -85,B 0,C 180,E1 -30926.519,E2 -30926.519} C_VEL
LIN {X 0,Y 45.421,Z 526.625,A -85,B 0,C 180,E1 -30938.173,E2 -30938.173} C_VEL
LIN {X 0,Y 58.215,Z 522.6,A -85,B 0,C 180,E1 -30944.96,E2 -30944.96} C_VEL
LIN {X 0,Y 71.499,Z 517.25,A -85,B 0,C 180,E1 -30949.391,E2 -30949.391} C_VEL
LIN {X 0,Y 85.074,Z 510.413,A -85,B 0,C 180,E1 -30952.432,E2 -30952.432} C_VEL
LIN {X 0,Y 91.922,Z 506.373,A -85,B 0,C 180,E1 -30953.664,E2 -30953.664} C_VEL
LIN {X 0,Y 93.808,Z 505.144,A -85,B 0,C 180,E1 -30954.748,E2 -30954.748} C_VEL
LIN {X 0,Y 94.769,Z 504.702,A -85,B 0,C 180,E1 -30960,E2 -30960} C_VEL
LIN {X 0,Y 94.267,Z 505.185,A -85,B 0,C 180,E1 -30961.709,E2 -30961.709} C_VEL
LIN {X 0,Y 92.997,Z 506.19,A -85,B 0,C 180,E1 -30963.321,E2 -30963.321} C_VEL
LIN {X 0,Y 85.466,Z 510.786,A -85,B 0,C 180,E1 -30964.487,E2 -30964.487} C_VEL
LIN {X 0,Y 80.309,Z 513.615,A -85,B 0,C 180,E1 -30964.916,E2 -30964.916} C_VEL
LIN {X 0,Y 71.321,Z 517.778,A -85,B 0,C 180,E1 -30964.4,E2 -30964.4} C_VEL
LIN {X 0,Y 62.12,Z 521.496,A -85,B 0,C 180,E1 -30963.789,E2 -30963.789} C_VEL
LIN {X 0,Y 56.609,Z 523.475,A -85,B 0,C 180,E1 -30964.424,E2 -30964.424} C_VEL
LIN {X 0,Y 41.149,Z 528.208,A -85,B 0,C 180,E1 -30969.833,E2 -30969.833} C_VEL
LIN {X 0,Y 29.553,Z 530.776,A -85,B 0,C 180,E1 -30977.984,E2 -30977.984} C_VEL
LIN {X 0,Y 17.996,Z 532.591,A -85,B 0,C 180,E1 -30998.657,E2 -30998.657} C_VEL
LIN {X 0,Y 13.039,Z 533.26,A -85,B 0,C 180,E1 -31050.013,E2 -31050.013} C_VEL
LIN {X 0,Y 18.003,Z 532.568,A -85,B 0,C 180,E1 -31101.344,E2 -31101.344} C_VEL
LIN {X 0,Y 29.549,Z 530.719,A -85,B 0,C 180,E1 -31122.076,E2 -31122.076} C_VEL
LIN {X 0,Y 42.704,Z 527.697,A -85,B 0,C 180,E1 -31130.94,E2 -31130.94} C_VEL
LIN {X 0,Y 56.398,Z 523.444,A -85,B 0,C 180,E1 -31135.53,E2 -31135.53} C_VEL
LIN {X 0,Y 70.314,Z 517.847,A -85,B 0,C 180,E1 -31138.29,E2 -31138.29} C_VEL
LIN {X 0,Y 84.34,Z 510.75,A -85,B 0,C 180,E1 -31140.231,E2 -31140.231} C_VEL
LIN {X 0,Y 87.022,Z 509.191,A -85,B 0,C 180,E1 -31140.522,E2 -31140.522} C_VEL
LIN {X 0,Y 88.345,Z 508.374,A -85,B 0,C 180,E1 -31141.477,E2 -31141.477} C_VEL
LIN {X 0,Y 87.103,Z 509.042,A -85,B 0,C 180,E1 -31142.519,E2 -31142.519} C_VEL
LIN {X 0,Y 74.015,Z 515.852,A -85,B 0,C 180,E1 -31144.401,E2 -31144.401} C_VEL
LIN {X 0,Y 60.222,Z 521.613,A -85,B 0,C 180,E1 -31147.249,E2 -31147.249} C_VEL
LIN {X 0,Y 50.027,Z 525.012,A -85,B 0,C 180,E1 -31150.438,E2 -31150.438} C_VEL
LIN {X 0,Y 36.748,Z 528.441,A -85,B 0,C 180,E1 -31156.997,E2 -31156.997} C_VEL
LIN {X 0,Y 24.366,Z 530.688,A -85,B 0,C 180,E1 -31170.069,E2 -31170.069} C_VEL
LIN {X 0,Y 15.032,Z 531.813,A -85,B 0,C 180,E1 -31202.113,E2 -31202.113} C_VEL
LIN {X 0,Y 13.522,Z 531.958,A -85,B 0,C 180,E1 -31229.987,E2 -31229.987} C_VEL
LIN {X 0,Y 19.015,Z 531.413,A -85,B 0,C 180,E1 -31277.651,E2 -31277.651} C_VEL
LIN {X 0,Y 30.361,Z 529.768,A -85,B 0,C 180,E1 -31297.794,E2 -31297.794} C_VEL
LIN {X 0,Y 43.282,Z 526.974,A -85,B 0,C 180,E1 -31306.953,E2 -31306.953} C_VEL
LIN {X 0,Y 56.783,Z 522.949,A -85,B 0,C 180,E1 -31311.934,E2 -31311.934} C_VEL
LIN {X 0,Y 70.537,Z 517.597,A -85,B 0,C 180,E1 -31315.077,E2 -31315.077} C_VEL
LIN {X 0,Y 84.432,Z 510.76,A -85,B 0,C 180,E1 -31317.226,E2 -31317.226} C_VEL
LIN {X 0,Y 87.149,Z 509.21,A -85,B 0,C 180,E1 -31317.58,E2 -31317.58} C_VEL
LIN {X 0,Y 88.405,Z 508.532,A -85,B 0,C 180,E1 -31318.566,E2 -31318.566} C_VEL
LIN {X 0,Y 87.075,Z 509.35,A -85,B 0,C 180,E1 -31319.473,E2 -31319.473} C_VEL
LIN {X 0,Y 73.806,Z 516.354,A -85,B 0,C 180,E1 -31321.141,E2 -31321.141} C_VEL
LIN {X 0,Y 59.856,Z 522.284,A -85,B 0,C 180,E1 -31323.651,E2 -31323.651} C_VEL
LIN {X 0,Y 56.609,Z 523.475,A -85,B 0,C 180,E1 -31324.424,E2 -31324.424} C_VEL
LIN {X 0,Y 51.052,Z 525.334,A -85,B 0,C 180,E1 -31325.22,E2 -31325.22} C_VEL
LIN {X 0,Y 41.476,Z 527.865,A -85,B 0,C 180,E1 -31324.64,E2 -31324.64} C_VEL
LIN {X 0,Y 33.703,Z 529.463,A -85,B 0,C 180,E1 -31323.714,E2 -31323.714} C_VEL
LIN {X 0,Y 27.868,Z 530.481,A -85,B 0,C 180,E1 -31324.238,E2 -31324.238} C_VEL
LIN {X 0,Y 25.951,Z 530.762,A -85,B 0,C 180,E1 -31325.024,E2 -31325.024} C_VEL
LIN {X 0,Y 14.636,Z 532.241,A -85,B 0,C 180,E1 -31336.222,E2 -31336.222} C_VEL
LIN {X 0,Y 5.914,Z 532.911,A -85,B 0,C 180,E1 -31410.029,E2 -31410.029} C_VEL
LIN {X 0,Y 14.642,Z 532.217,A -85,B 0,C 180,E1 -31483.771,E2 -31483.771} C_VEL
LIN {X 0,Y 28.179,Z 530.366,A -85,B 0,C 180,E1 -31496.136,E2 -31496.136} C_VEL
LIN {X 0,Y 42.173,Z 527.344,A -85,B 0,C 180,E1 -31500.621,E2 -31500.621} C_VEL
LIN {X 0,Y 49.225,Z 525.379,A -85,B 0,C 180,E1 -31501.86,E2 -31501.86} C_VEL
LIN {X 0,Y 49.237,Z 525.362,A -85,B 0,C 180,E1 -31502.258,E2 -31502.258} C_VEL
LIN {X 0,Y 35.327,Z 528.791,A -85,B 0,C 180,E1 -31505.858,E2 -31505.858} C_VEL
LIN {X 0,Y 21.693,Z 531.037,A -85,B 0,C 180,E1 -31513.571,E2 -31513.571} C_VEL
LIN {X 0,Y 9.364,Z 532.161,A -85,B 0,C 180,E1 -31541.337,E2 -31541.337} C_VEL
LIN {X 0,Y 6.449,Z 532.305,A -85,B 0,C 180,E1 -31589.974,E2 -31589.974} C_VEL
LIN {X 0,Y 15.164,Z 531.762,A -85,B 0,C 180,E1 -31657.934,E2 -31657.934} C_VEL
LIN {X 0,Y 28.443,Z 530.117,A -85,B 0,C 180,E1 -31671.216,E2 -31671.216} C_VEL
LIN {X 0,Y 42.249,Z 527.321,A -85,B 0,C 180,E1 -31676.392,E2 -31676.392} C_VEL
LIN {X 0,Y 49.228,Z 525.464,A -85,B 0,C 180,E1 -31677.848,E2 -31677.848} C_VEL
LIN {X 0,Y 49.219,Z 525.477,A -85,B 0,C 180,E1 -31678.15,E2 -31678.15} C_VEL
LIN {X 0,Y 35.146,Z 529.078,A -85,B 0,C 180,E1 -31681.273,E2 -31681.273} C_VEL
LIN {X 0,Y 25.951,Z 530.762,A -85,B 0,C 180,E1 -31685.024,E2 -31685.024} C_VEL
LIN {X 0,Y 24.294,Z 532.74,A -85,B 0,C 180,E1 -31685.97,E2 -31685.97} C_VEL
LIN {X 0,Y 24.294,Z 600,A -85,B 0,C 180,E1 -31685.97,E2 -31685.97} C_VEL
LIN {X 0,Y 24.294,Z 600,A -85,B 0,C 180,E1 -31685.97,E2 -31685.97}

QRS_NEXT_CUT()

QRS_NEXT()
QRS_HOME()

END
